FUNCTION_BLOCK InfluentActuators (* CAT Function Block Type *)
  (* Standard: 61499-2 *)
  (* Version 0.0, 6/13/2026, Schneider Electric, template *)
  PACKAGE SE.Nereda;
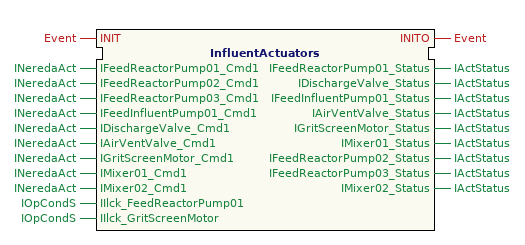
  EVENT_INPUT
    INIT;
  END_EVENT
  EVENT_OUTPUT
    INITO;
  END_EVENT
  SOCKETS
    IFeedReactorPump01_Cmd1 : INeredaAct;
    IFeedReactorPump02_Cmd1 : INeredaAct;
    IFeedReactorPump03_Cmd1 : INeredaAct;
    IFeedInfluentPump01_Cmd1 : INeredaAct;
    IDischargeValve_Cmd1 : INeredaAct;
    IAirVentValve_Cmd1 : INeredaAct;
    IGritScreenMotor_Cmd1 : INeredaAct;
    IMixer01_Cmd1 : INeredaAct;
    IMixer02_Cmd1 : INeredaAct;
    IIlck_FeedReactorPump01 : IOpCondS; (* Condition summary chain input from upstream blocks *)
    IIlck_GritScreenMotor : IOpCondS; (* Condition summary chain input from upstream blocks *)
  END_SOCKETS
  PLUGS
    IFeedReactorPump01_Status : IActStatus;
    IDischargeValve_Status : IActStatus;
    IFeedInfluentPump01_Status : IActStatus;
    IAirVentValve_Status : IActStatus;
    IGritScreenMotor_Status : IActStatus;
    IMixer01_Status : IActStatus;
    IFeedReactorPump02_Status : IActStatus;
    IFeedReactorPump03_Status : IActStatus;
    IMixer02_Status : IActStatus;
  END_PLUGS
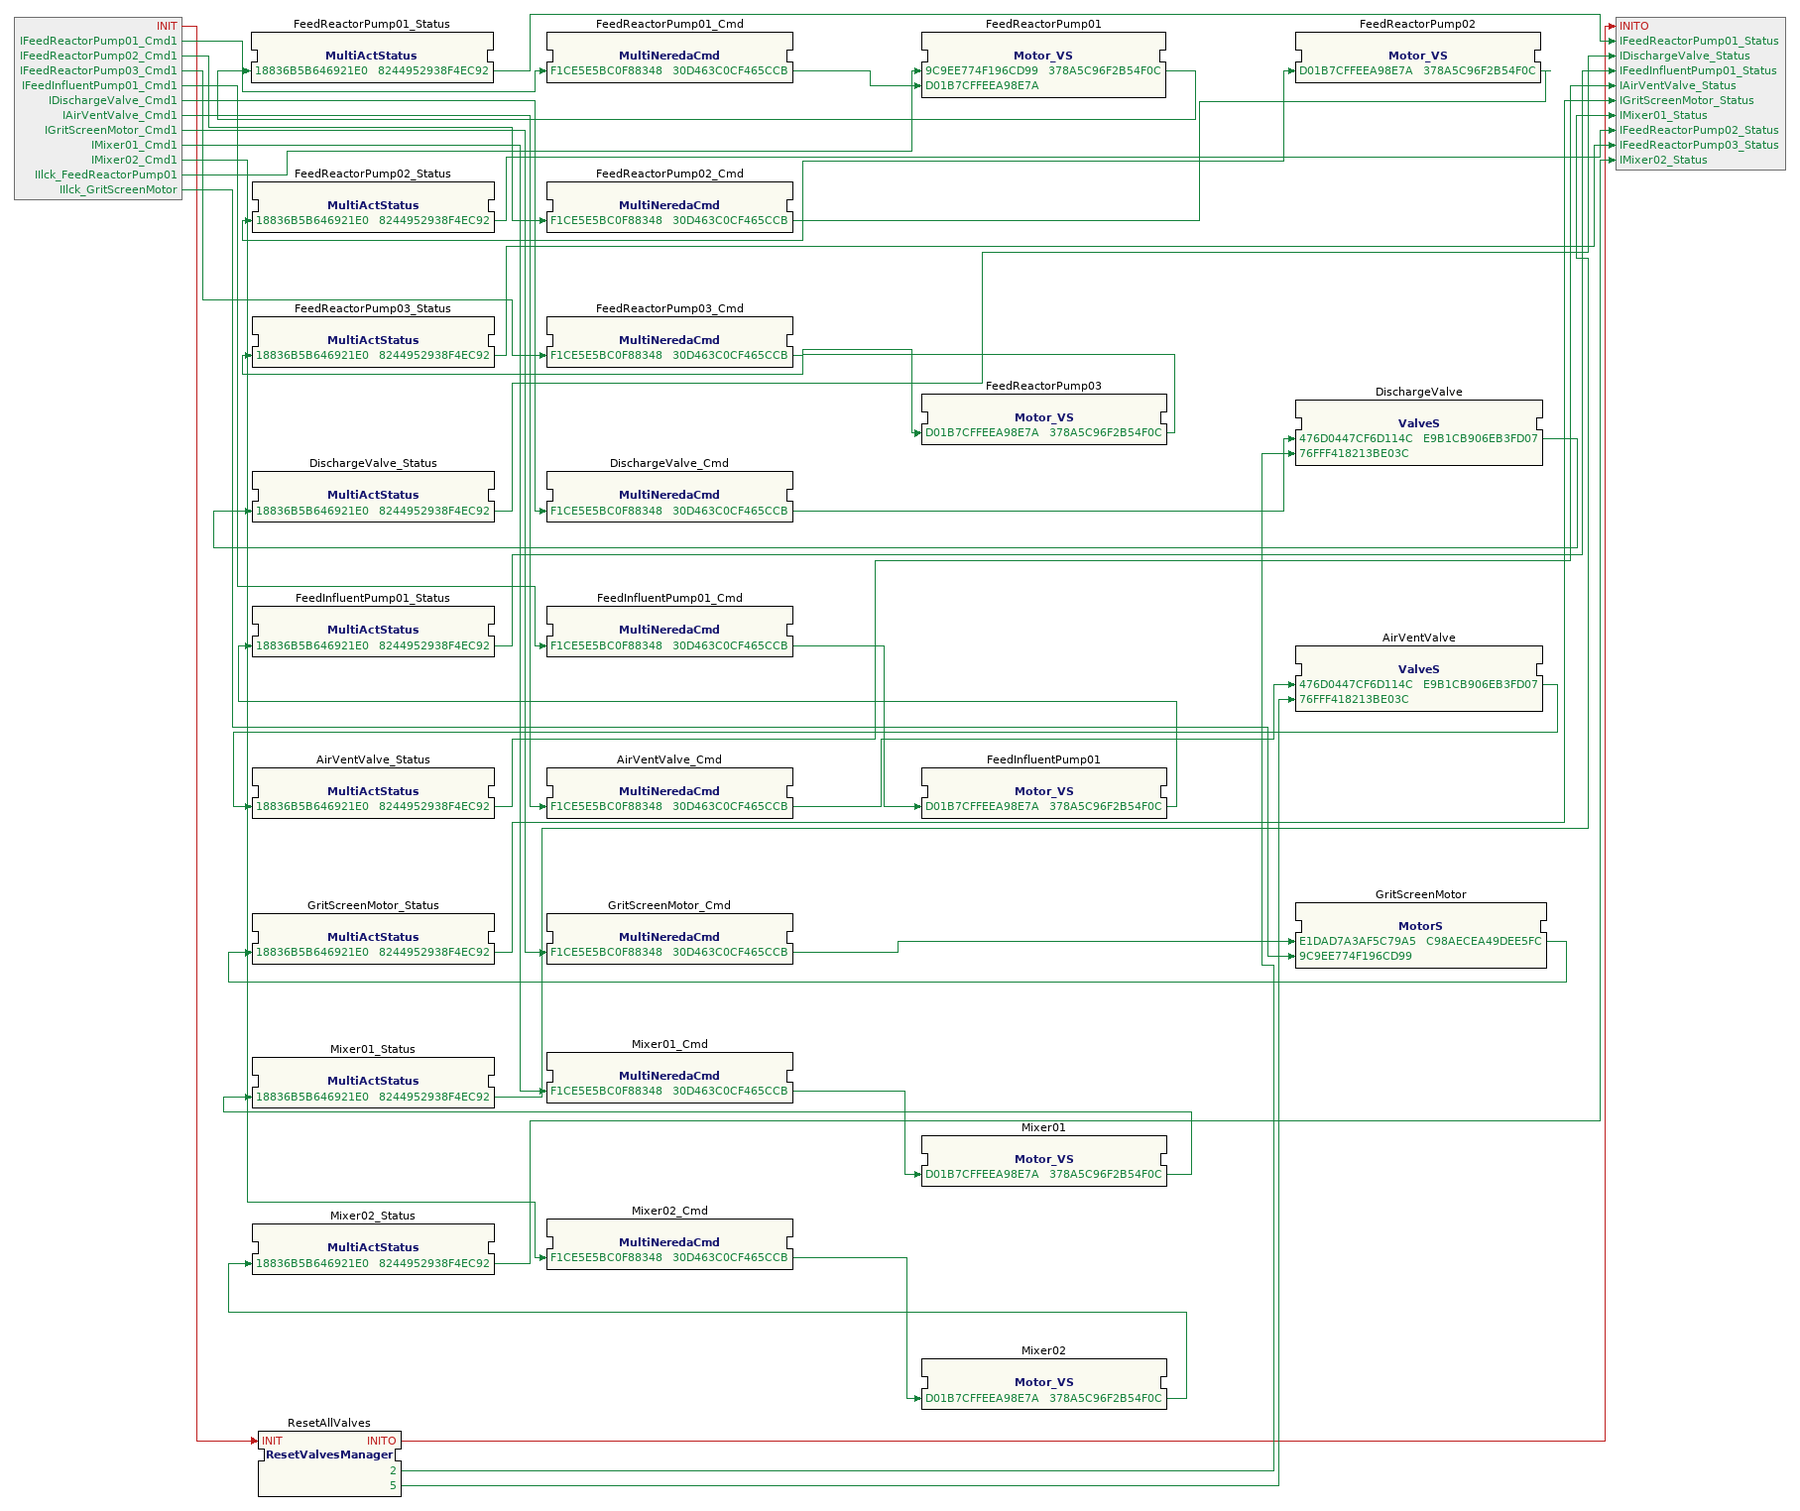
  (* 01 - FUNCTIONNAL INPUT INTERFACE *)
  (* 00 - INITIALIZATION *)
  (* 05 - LOGIC *)
  (* 06 - HMI INTERFACE *)
  (* 03 - FIELD INTERFACE *)
  (* 02 - FUNCTIONNAL OUTPUT INTERFACE *)
  (* Actuators Status *)
  (* 04 - CHILDREN *)
  (* 4A - TYPICALS *)
  (* Actuators Command *)
  (* Reset All Actuators *)
  FBS
    ResetAllValves : ResetValvesManager;
    FeedReactorPump01_Status : MultiActStatus;
    DischargeValve_Status : MultiActStatus;
    FeedInfluentPump01_Status : MultiActStatus;
    AirVentValve_Status : MultiActStatus;
    GritScreenMotor_Status : MultiActStatus;
    FeedReactorPump01_Cmd : MultiNeredaCmd;
    DischargeValve_Cmd : MultiNeredaCmd;
    FeedInfluentPump01_Cmd : MultiNeredaCmd;
    GritScreenMotor_Cmd : MultiNeredaCmd;
    AirVentValve_Cmd : MultiNeredaCmd;
    FeedReactorPump01 : Motor_VS;
    FeedInfluentPump01 : Motor_VS;
    DischargeValve : ValveS;
    AirVentValve : ValveS;
    GritScreenMotor : MotorS;
    Mixer01_Cmd : MultiNeredaCmd;
    Mixer01_Status : MultiActStatus;
    Mixer01 : Motor_VS;
    Mixer02 : Motor_VS;
    Mixer02_Cmd : MultiNeredaCmd;
    Mixer02_Status : MultiActStatus;
    FeedReactorPump02 : Motor_VS;
    FeedReactorPump03 : Motor_VS;
    FeedReactorPump02_Status : MultiActStatus;
    FeedReactorPump02_Cmd : MultiNeredaCmd;
    FeedReactorPump03_Status : MultiActStatus;
    FeedReactorPump03_Cmd : MultiNeredaCmd;
  END_FBS
  EVENT_CONNECTIONS
    INIT TO ResetAllValves.INIT;
    ResetAllValves.INITO TO INITO;
  END_CONNECTIONS
  ADAPTER_CONNECTIONS
    IFeedReactorPump01_Cmd1 TO FeedReactorPump01_Cmd.F1CE5E5BC0F88348;
    IDischargeValve_Cmd1 TO DischargeValve_Cmd.F1CE5E5BC0F88348;
    IFeedInfluentPump01_Cmd1 TO FeedInfluentPump01_Cmd.F1CE5E5BC0F88348;
    IAirVentValve_Cmd1 TO AirVentValve_Cmd.F1CE5E5BC0F88348;
    IGritScreenMotor_Cmd1 TO GritScreenMotor_Cmd.F1CE5E5BC0F88348;
    IMixer01_Cmd1 TO Mixer01_Cmd.F1CE5E5BC0F88348;
    IIlck_FeedReactorPump01 TO FeedReactorPump01.9C9EE774F196CD99;
    FeedReactorPump01_Cmd.30D463C0CF465CCB TO FeedReactorPump01.D01B7CFFEEA98E7A;
    DischargeValve_Cmd.30D463C0CF465CCB TO DischargeValve.476D0447CF6D114C;
    FeedInfluentPump01_Cmd.30D463C0CF465CCB TO FeedInfluentPump01.D01B7CFFEEA98E7A;
    AirVentValve_Cmd.30D463C0CF465CCB TO AirVentValve.476D0447CF6D114C;
    GritScreenMotor_Cmd.30D463C0CF465CCB TO GritScreenMotor.E1DAD7A3AF5C79A5;
    Mixer01_Cmd.30D463C0CF465CCB TO Mixer01.D01B7CFFEEA98E7A;
    FeedReactorPump01.378A5C96F2B54F0C TO FeedReactorPump01_Status.18836B5B646921E0;
    DischargeValve.E9B1CB906EB3FD07 TO DischargeValve_Status.18836B5B646921E0;
    FeedInfluentPump01.378A5C96F2B54F0C TO FeedInfluentPump01_Status.18836B5B646921E0;
    AirVentValve.E9B1CB906EB3FD07 TO AirVentValve_Status.18836B5B646921E0;
    GritScreenMotor.C98AECEA49DEE5FC TO GritScreenMotor_Status.18836B5B646921E0;
    Mixer01.378A5C96F2B54F0C TO Mixer01_Status.18836B5B646921E0;
    FeedReactorPump01_Status.8244952938F4EC92 TO IFeedReactorPump01_Status;
    DischargeValve_Status.8244952938F4EC92 TO IDischargeValve_Status;
    FeedInfluentPump01_Status.8244952938F4EC92 TO IFeedInfluentPump01_Status;
    AirVentValve_Status.8244952938F4EC92 TO IAirVentValve_Status;
    GritScreenMotor_Status.8244952938F4EC92 TO IGritScreenMotor_Status;
    Mixer01_Status.8244952938F4EC92 TO IMixer01_Status;
    ResetAllValves.2 TO DischargeValve.76FFF418213BE03C;
    ResetAllValves.5 TO AirVentValve.76FFF418213BE03C;
    IIlck_GritScreenMotor TO GritScreenMotor.9C9EE774F196CD99;
    Mixer02_Cmd.30D463C0CF465CCB TO Mixer02.D01B7CFFEEA98E7A;
    Mixer02.378A5C96F2B54F0C TO Mixer02_Status.18836B5B646921E0;
    IFeedReactorPump02_Cmd1 TO FeedReactorPump02_Cmd.F1CE5E5BC0F88348;
    IFeedReactorPump03_Cmd1 TO FeedReactorPump03_Cmd.F1CE5E5BC0F88348;
    FeedReactorPump02.378A5C96F2B54F0C TO FeedReactorPump02_Status.18836B5B646921E0;
    FeedReactorPump03.378A5C96F2B54F0C TO FeedReactorPump03_Status.18836B5B646921E0;
    FeedReactorPump02_Cmd.30D463C0CF465CCB TO FeedReactorPump02.D01B7CFFEEA98E7A;
    FeedReactorPump03_Cmd.30D463C0CF465CCB TO FeedReactorPump03.D01B7CFFEEA98E7A;
    FeedReactorPump02_Status.8244952938F4EC92 TO IFeedReactorPump02_Status;
    FeedReactorPump03_Status.8244952938F4EC92 TO IFeedReactorPump03_Status;
    IMixer02_Cmd1 TO Mixer02_Cmd.F1CE5E5BC0F88348;
    Mixer02_Status.8244952938F4EC92 TO IMixer02_Status;
  END_CONNECTIONS
END_FUNCTION_BLOCK
